PROGRAM MAIN
VAR
	Demo : FB_Demo;
END_VAR

Demo();

END_PROGRAM

(* stored: Version 1.1.0.1, ProductVersion 3.1.4024.12
   POU MAIN: Id {a2110135-111d-486c-a926-541f4e1370f7}, SpecialFunc None *)
